// TIA Portal V17 export
// export: Created 2025-06-26T06:49:16.0096104Z, ExportSetting WithDefaults, DisplayName Totally Integrated Automation Portal, DisplayVersion V17 Update 8, DisplayName TIA Portal Openness, DisplayVersion V17 Update 8, DisplayName TIA Portal Version Control Interface, DisplayVersion V17, DisplayName STEP 7 Professional, DisplayVersion V17 Update 8, DisplayName STEP 7 Safety, DisplayVersion V17 Update 6, DisplayName WinCC Advanced, DisplayVersion V17 Update 8
FUNCTION_BLOCK "fbDigitalAlarm"   // FB47, FBD
{ S7_Optimized_Access := 'TRUE' }
VERSION : 0.1
// stored: AutoNumber true, IsIECCheckEnabled false, IsRetainMemResEnabled false, MemoryReserve 0, SetENOAutomatically false, UDAEnableTagReadback false
   VAR_INPUT
      bInput : Bool;
      bAckAll : Bool;
      bEnable : Bool;
   END_VAR
   VAR_IN_OUT
      sTag : "stDigitalAlarm";
   END_VAR
   VAR
      Alarm : "fbAlarm";
   END_VAR
BEGIN

REGION Network 1
   // The Enables are ANDed together to allow the struct one to act as a disable bit
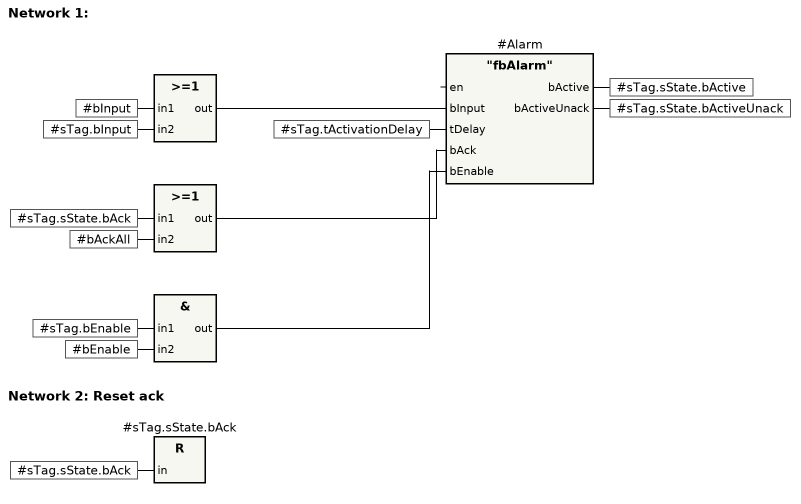
   #Alarm(bInput := #bInput OR #sTag.bInput,   // "fbAlarm"
          tDelay := #sTag.tActivationDelay,
          bAck := #sTag.sState.bAck OR #bAckAll,
          bEnable := #sTag.bEnable AND #bEnable,
          bActive => #sTag.sState.bActive,
          bActiveUnack => #sTag.sState.bActiveUnack);
END_REGION

REGION Network 2: Reset ack
   IF #sTag.sState.bAck THEN #sTag.sState.bAck := FALSE; END_IF;
END_REGION
END_FUNCTION_BLOCK
